(* IEC 61131-3 sources: CodesysTest/alpha/export/Pro18_1174_CodesysDriver.dev/Plc Logic/Application/Motors/Applied Motion/FB_AppliedMotionStepServoEIPBase.pou/HomeRequired.prop, 1 file *)

(* ---- Set.pm.st ---- *)
(*#-#-#-#-#-#-#-#-#-#---Declaration---#-#-#-#-#-#-#-#-#-#-#-#-#*)

VAR
END_VAR
(*#-#-#-#-#-#-#-#-#-#---Implementation---#-#-#-#-#-#-#-#-#-#-#-#-#*)

homeRequiredIndication := HomeRequired;
